TYPE ST_AC_Swing :
STRUCT
	HorizOn: BOOL;
	HorizOff: BOOL;
	VertiOn: BOOL;
	VertiOff: BOOL;
END_STRUCT
END_TYPE

(* stored: Version 1.1.0.1, ProductVersion 3.1.4024.12
   DUT ST_AC_Swing: Id {cd383b55-d960-4eb7-9476-01201f6cb636} *)
